// TIA Portal V20 export
DATA_BLOCK "Instance_FB_Digital_Inputs_DB"   // DB101
// stored: AutoNumber false, InstanceOfName FB_Digital_Inputs, InstanceOfType FB
"FB_Digital_Inputs"
   // VAR_INPUT
   //    I_Button_Start_Approve : Bool;
   //    I_Digital_Input_1 : Bool;
   //    I_Digital_Input_2 : Bool;
   //    I_Digital_Input_3 : Bool;
   //    I_Digital_Input_4 : Bool;
   //    I_Digital_Input_5 : Bool;
   // END_VAR
   // VAR_OUTPUT
   //    DB_Button_Start_Approve : Bool;
   //    DB_Digital_Input_1 : Bool;
   //    DB_Digital_Input_2 : Bool;
   //    DB_Digital_Input_3 : Bool;
   //    DB_Digital_Input_4 : Bool;
   //    DB_Digital_Input_5 : Bool;
   // END_VAR
BEGIN
END_DATA_BLOCK
